PROGRAM myCNC_Call_Roll
VAR
END_VAR

END_PROGRAM

(* stored: Version 1.1.0.1, ProductVersion 3.1.4024.11
   POU myCNC_Call_Roll: Id {2378917e-6b18-4210-8389-0d29887bc909}, SpecialFunc None *)
